Staubli VAL3: registerSetting.pgx

public program registerSetting(settingType& setting_, num index_)
begin
  switch index_
    case 0
      setting_.label="Safety Distance"
      setting_.varName=$getName(nMouldAreaZone)
      setting_.sType="num"
      setting_.nValue=0
      setting_.format="5.0"
      setting_.sDescription="Safety Distance to Mould"
      setting_.parentName="IMM"+toString("0.0",moduleIndex)
    break

    case 1
      setting_.label="IMM Type"
      setting_.varName="nImmType"
      setting_.sType="num"
      setting_.nValue=0
      setting_.sDescription="This setting changes the behaviour of the IMM: 0: Netstal, 1: Neggri Bossi"
      setting_.parentName="IMM"+toString("0.0",moduleIndex)
    break

    case 2
      setting_.label="Monitor Mould Area"
      setting_.varName="bMonitorArea"
      setting_.sType="bool"
      setting_.bValue=true
      setting_.sDescription=""
      setting_.parentName="IMM"+toString("0.0",moduleIndex)
    break
  endSwitch
end
